// TIA Portal V20 export
FUNCTION "Fnet06" : Void   // FC138, LAD
// stored: Namespace Unit1, SetENOAutomatically false
BEGIN

REGION Network 1: Part Pass
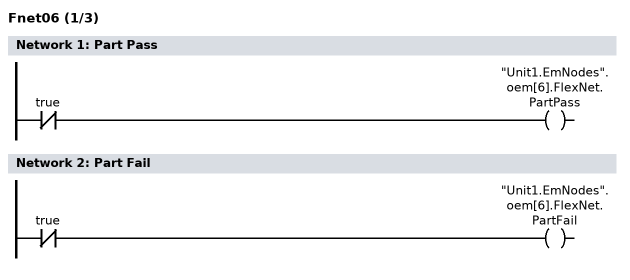
   RUNG wire#powerrail
      I_Contact( true )
      Coil( "Unit1.EmNodes".oem[6].FlexNet.PartPass )
   END_RUNG
   // the same network as SCL:
   "Unit1.EmNodes".oem[6].FlexNet.PartPass := NOT true;
END_REGION

REGION Network 2: Part Fail
   RUNG wire#powerrail
      I_Contact( true )
      Coil( "Unit1.EmNodes".oem[6].FlexNet.PartFail )
   END_RUNG
   // the same network as SCL:
   "Unit1.EmNodes".oem[6].FlexNet.PartFail := NOT true;
END_REGION

REGION Network 3: Pun, GM Part Number, Optional Data, Tracking ID, Tracking ID Attribute, and Data Ready
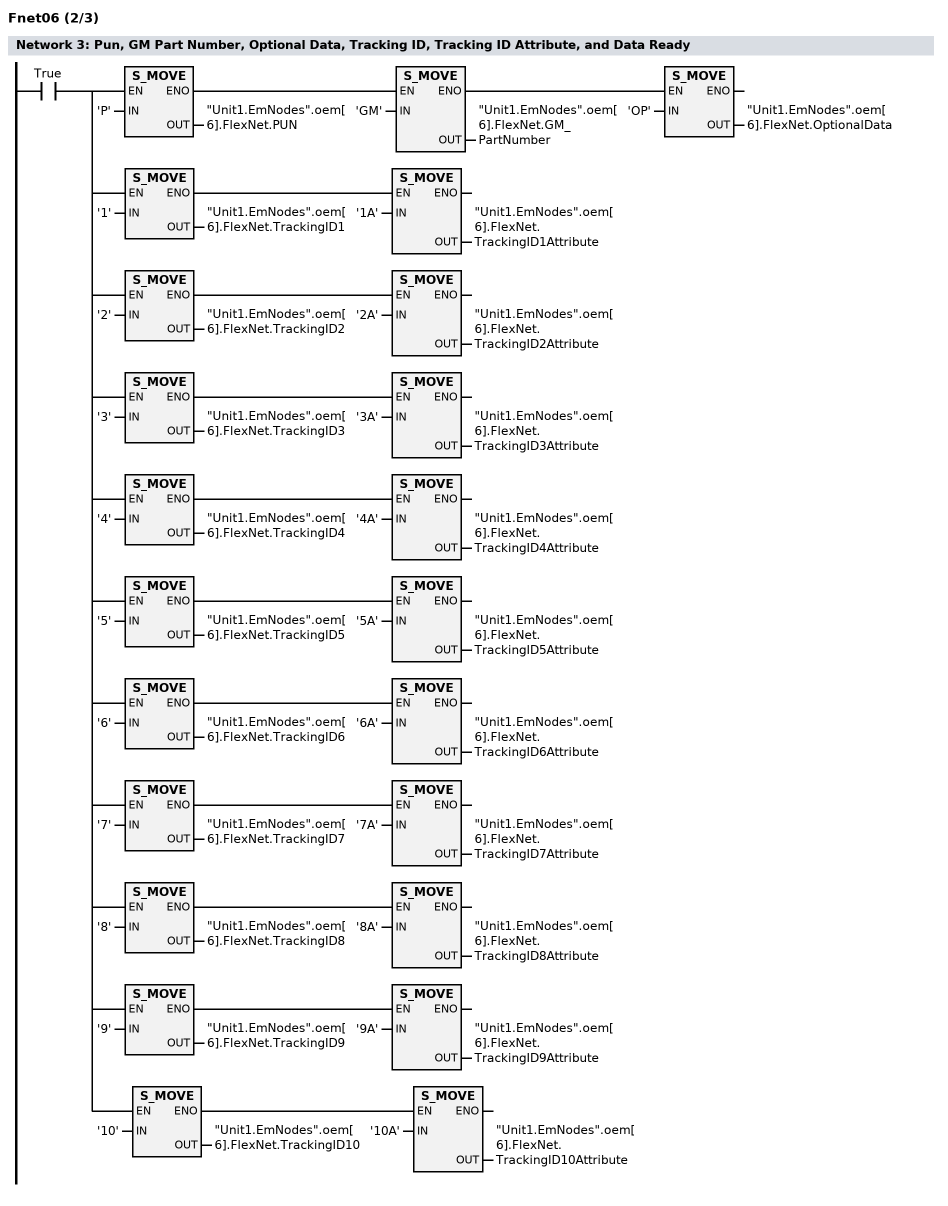
   RUNG wire#powerrail
      Contact( True )
      wire#w1
      S_Move(in := 'P', out => "Unit1.EmNodes".oem[6].FlexNet.PUN)
      S_Move(in := 'GM', out => "Unit1.EmNodes".oem[6].FlexNet.GM_PartNumber)
      S_Move(in := 'OP', out => "Unit1.EmNodes".oem[6].FlexNet.OptionalData)
   END_RUNG
   RUNG wire#w1
      S_Move(in := '1', out => "Unit1.EmNodes".oem[6].FlexNet.TrackingID1)
      S_Move(in := '1A', out => "Unit1.EmNodes".oem[6].FlexNet.TrackingID1Attribute)
   END_RUNG
   RUNG wire#w1
      S_Move(in := '2', out => "Unit1.EmNodes".oem[6].FlexNet.TrackingID2)
      S_Move(in := '2A', out => "Unit1.EmNodes".oem[6].FlexNet.TrackingID2Attribute)
   END_RUNG
   RUNG wire#w1
      S_Move(in := '3', out => "Unit1.EmNodes".oem[6].FlexNet.TrackingID3)
      S_Move(in := '3A', out => "Unit1.EmNodes".oem[6].FlexNet.TrackingID3Attribute)
   END_RUNG
   RUNG wire#w1
      S_Move(in := '4', out => "Unit1.EmNodes".oem[6].FlexNet.TrackingID4)
      S_Move(in := '4A', out => "Unit1.EmNodes".oem[6].FlexNet.TrackingID4Attribute)
   END_RUNG
   RUNG wire#w1
      S_Move(in := '5', out => "Unit1.EmNodes".oem[6].FlexNet.TrackingID5)
      S_Move(in := '5A', out => "Unit1.EmNodes".oem[6].FlexNet.TrackingID5Attribute)
   END_RUNG
   RUNG wire#w1
      S_Move(in := '6', out => "Unit1.EmNodes".oem[6].FlexNet.TrackingID6)
      S_Move(in := '6A', out => "Unit1.EmNodes".oem[6].FlexNet.TrackingID6Attribute)
   END_RUNG
   RUNG wire#w1
      S_Move(in := '7', out => "Unit1.EmNodes".oem[6].FlexNet.TrackingID7)
      S_Move(in := '7A', out => "Unit1.EmNodes".oem[6].FlexNet.TrackingID7Attribute)
   END_RUNG
   RUNG wire#w1
      S_Move(in := '8', out => "Unit1.EmNodes".oem[6].FlexNet.TrackingID8)
      S_Move(in := '8A', out => "Unit1.EmNodes".oem[6].FlexNet.TrackingID8Attribute)
   END_RUNG
   RUNG wire#w1
      S_Move(in := '9', out => "Unit1.EmNodes".oem[6].FlexNet.TrackingID9)
      S_Move(in := '9A', out => "Unit1.EmNodes".oem[6].FlexNet.TrackingID9Attribute)
   END_RUNG
   RUNG wire#w1
      S_Move(in := '10', out => "Unit1.EmNodes".oem[6].FlexNet.TrackingID10)
      S_Move(in := '10A', out => "Unit1.EmNodes".oem[6].FlexNet.TrackingID10Attribute)
   END_RUNG
   // the same network as SCL:
   IF True THEN
       "Unit1.EmNodes".oem[6].FlexNet.PUN := 'P';
       "Unit1.EmNodes".oem[6].FlexNet.GM_PartNumber := 'GM';
       "Unit1.EmNodes".oem[6].FlexNet.OptionalData := 'OP';
       "Unit1.EmNodes".oem[6].FlexNet.TrackingID1 := '1';
       "Unit1.EmNodes".oem[6].FlexNet.TrackingID1Attribute := '1A';
       "Unit1.EmNodes".oem[6].FlexNet.TrackingID2 := '2';
       "Unit1.EmNodes".oem[6].FlexNet.TrackingID2Attribute := '2A';
       "Unit1.EmNodes".oem[6].FlexNet.TrackingID3 := '3';
       "Unit1.EmNodes".oem[6].FlexNet.TrackingID3Attribute := '3A';
       "Unit1.EmNodes".oem[6].FlexNet.TrackingID4 := '4';
       "Unit1.EmNodes".oem[6].FlexNet.TrackingID4Attribute := '4A';
       "Unit1.EmNodes".oem[6].FlexNet.TrackingID5 := '5';
       "Unit1.EmNodes".oem[6].FlexNet.TrackingID5Attribute := '5A';
       "Unit1.EmNodes".oem[6].FlexNet.TrackingID6 := '6';
       "Unit1.EmNodes".oem[6].FlexNet.TrackingID6Attribute := '6A';
       "Unit1.EmNodes".oem[6].FlexNet.TrackingID7 := '7';
       "Unit1.EmNodes".oem[6].FlexNet.TrackingID7Attribute := '7A';
       "Unit1.EmNodes".oem[6].FlexNet.TrackingID8 := '8';
       "Unit1.EmNodes".oem[6].FlexNet.TrackingID8Attribute := '8A';
       "Unit1.EmNodes".oem[6].FlexNet.TrackingID9 := '9';
       "Unit1.EmNodes".oem[6].FlexNet.TrackingID9Attribute := '9A';
       "Unit1.EmNodes".oem[6].FlexNet.TrackingID10 := '10';
       "Unit1.EmNodes".oem[6].FlexNet.TrackingID10Attribute := '10A';
   END_IF;
END_REGION

REGION Network 4: Part Fail
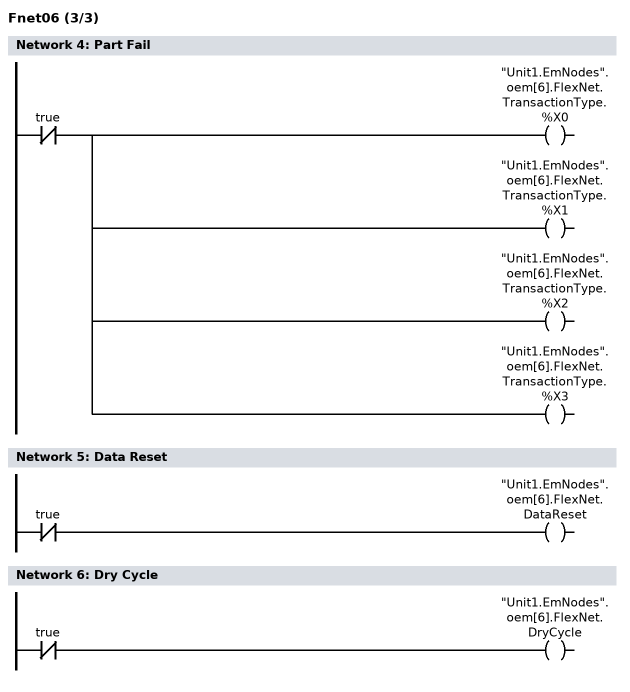
   RUNG wire#powerrail
      I_Contact( true )
      wire#w1
      Coil( "Unit1.EmNodes".oem[6].FlexNet.TransactionType.%X0 )
   END_RUNG
   RUNG wire#w1
      Coil( "Unit1.EmNodes".oem[6].FlexNet.TransactionType.%X1 )
   END_RUNG
   RUNG wire#w1
      Coil( "Unit1.EmNodes".oem[6].FlexNet.TransactionType.%X2 )
   END_RUNG
   RUNG wire#w1
      Coil( "Unit1.EmNodes".oem[6].FlexNet.TransactionType.%X3 )
   END_RUNG
   // the same network as SCL:
   "Unit1.EmNodes".oem[6].FlexNet.TransactionType.%X0 := NOT true;
   "Unit1.EmNodes".oem[6].FlexNet.TransactionType.%X1 := NOT true;
   "Unit1.EmNodes".oem[6].FlexNet.TransactionType.%X2 := NOT true;
   "Unit1.EmNodes".oem[6].FlexNet.TransactionType.%X3 := NOT true;
END_REGION

REGION Network 5: Data Reset
   RUNG wire#powerrail
      I_Contact( true )
      Coil( "Unit1.EmNodes".oem[6].FlexNet.DataReset )
   END_RUNG
   // the same network as SCL:
   "Unit1.EmNodes".oem[6].FlexNet.DataReset := NOT true;
END_REGION

REGION Network 6: Dry Cycle
   RUNG wire#powerrail
      I_Contact( true )
      Coil( "Unit1.EmNodes".oem[6].FlexNet.DryCycle )
   END_RUNG
   // the same network as SCL:
   "Unit1.EmNodes".oem[6].FlexNet.DryCycle := NOT true;
END_REGION
END_FUNCTION
